PROGRAM PresenceSimulation
VAR
	
	fbWeeklyTimeSwitch	:FB_WeeklyTimeSwitch;
	fbSceneLight		:FB_IoT_Switch(P_IoT_Com.fbIoT_ComClient,0);
	CTU					:CTU;
	TON					:ARRAY[1..55] OF TON;
	TP					:ARRAY[1..55] OF TP;
	
	bAnwesenheit_Tag_1_aktivieren: BOOL;
	bAnwesenheit_Tag_2_aktivieren: BOOL;
	bAnwesenheit_Tag_3_aktivieren: BOOL;
	bAnwesenheit_Tag_4_aktivieren: BOOL;
	bAnwesenheit_Tag_5_aktivieren: BOOL;
	
	bAnwesenheit_1_Beleuchtung_1: BOOL;
	bAnwesenheit_1_Beleuchtung_2: BOOL;
	bAnwesenheit_1_Beleuchtung_3: BOOL;
	bAnwesenheit_1_Beleuchtung_4: BOOL;
	bAnwesenheit_1_Beleuchtung_5: BOOL;
	
	bAnwesenheit_2_Beleuchtung_1: BOOL;
	bAnwesenheit_2_Beleuchtung_2: BOOL;
	bAnwesenheit_2_Beleuchtung_3: BOOL;
	bAnwesenheit_2_Beleuchtung_4: BOOL;
	bAnwesenheit_2_Beleuchtung_5: BOOL;
	
	bAnwesenheit_3_Beleuchtung_1: BOOL;
	bAnwesenheit_3_Beleuchtung_2: BOOL;
	bAnwesenheit_3_Beleuchtung_3: BOOL;
	bAnwesenheit_3_Beleuchtung_4: BOOL;
	bAnwesenheit_3_Beleuchtung_5: BOOL;
	
	bAnwesenheit_4_Beleuchtung_1: BOOL;
	bAnwesenheit_4_Beleuchtung_2: BOOL;
	bAnwesenheit_4_Beleuchtung_3: BOOL;
	bAnwesenheit_4_Beleuchtung_4: BOOL;
	bAnwesenheit_4_Beleuchtung_5: BOOL;
	
	bAnwesenheit_5_Beleuchtung_1: BOOL;
	bAnwesenheit_5_Beleuchtung_2: BOOL;
	bAnwesenheit_5_Beleuchtung_3: BOOL;
	bAnwesenheit_5_Beleuchtung_4: BOOL;
	bAnwesenheit_5_Beleuchtung_5: BOOL;
END_VAR
VAR // added by the converter: edge detectors and wires of the graphical bodies
    _w1 : BOOL;
END_VAR

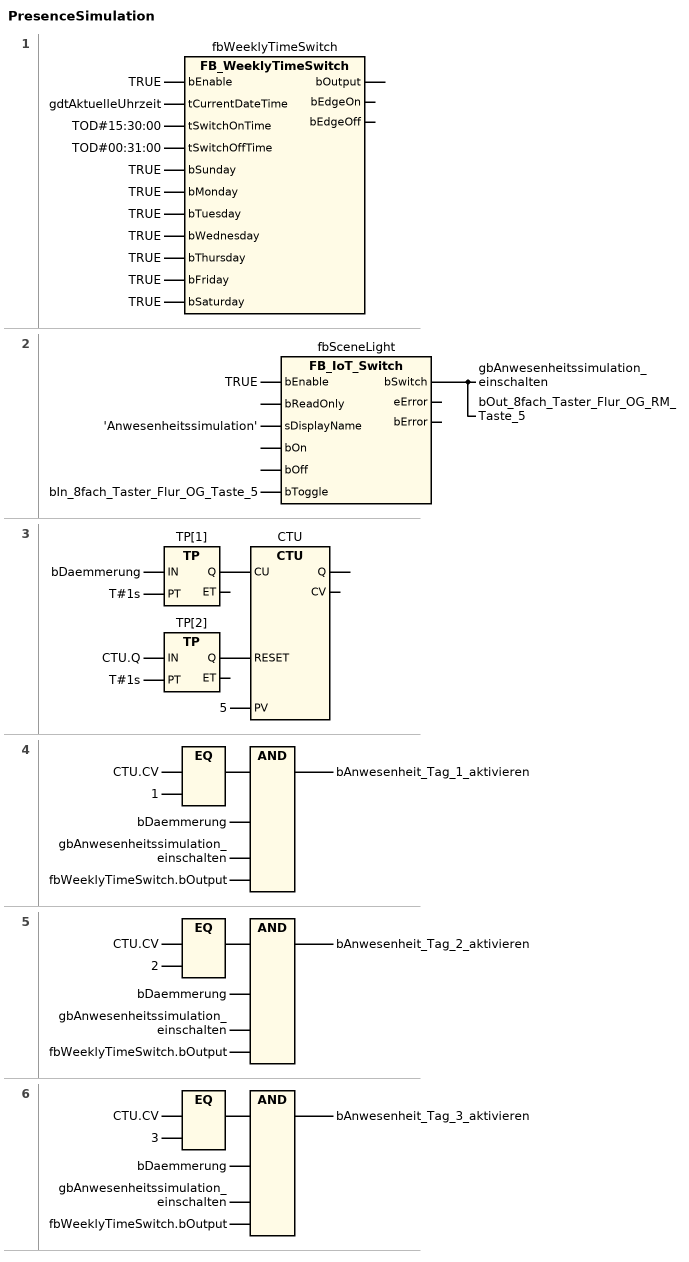
// NETWORK 1
fbWeeklyTimeSwitch(
    bEnable := TRUE,
    tCurrentDateTime := gdtAktuelleUhrzeit,
    tSwitchOnTime := TOD#15:30:00,
    tSwitchOffTime := TOD#00:31:00,
    bSunday := TRUE,
    bMonday := TRUE,
    bTuesday := TRUE,
    bWednesday := TRUE,
    bThursday := TRUE,
    bFriday := TRUE,
    bSaturday := TRUE); // FB_WeeklyTimeSwitch

// NETWORK 2
fbSceneLight(
    bEnable := TRUE,
    sDisplayName := 'Anwesenheitssimulation',
    bToggle := bIn_8fach_Taster_Flur_OG_Taste_5); // FB_IoT_Switch
gbAnwesenheitssimulation_einschalten := fbSceneLight.bSwitch;
bOut_8fach_Taster_Flur_OG_RM_Taste_5 := fbSceneLight.bSwitch;

// NETWORK 3
TP[1](IN := bDaemmerung, PT := T#1s); // TP
_w1 := TP[1].Q;
TP[2](IN := CTU.Q, PT := T#1s); // TP
CTU(CU := _w1, RESET := TP[2].Q, PV := 5);

// NETWORK 4
bAnwesenheit_Tag_1_aktivieren := CTU.CV = 1 AND bDaemmerung AND gbAnwesenheitssimulation_einschalten AND fbWeeklyTimeSwitch.bOutput;

// NETWORK 5
bAnwesenheit_Tag_2_aktivieren := CTU.CV = 2 AND bDaemmerung AND gbAnwesenheitssimulation_einschalten AND fbWeeklyTimeSwitch.bOutput;

// NETWORK 6
bAnwesenheit_Tag_3_aktivieren := CTU.CV = 3 AND bDaemmerung AND gbAnwesenheitssimulation_einschalten AND fbWeeklyTimeSwitch.bOutput;

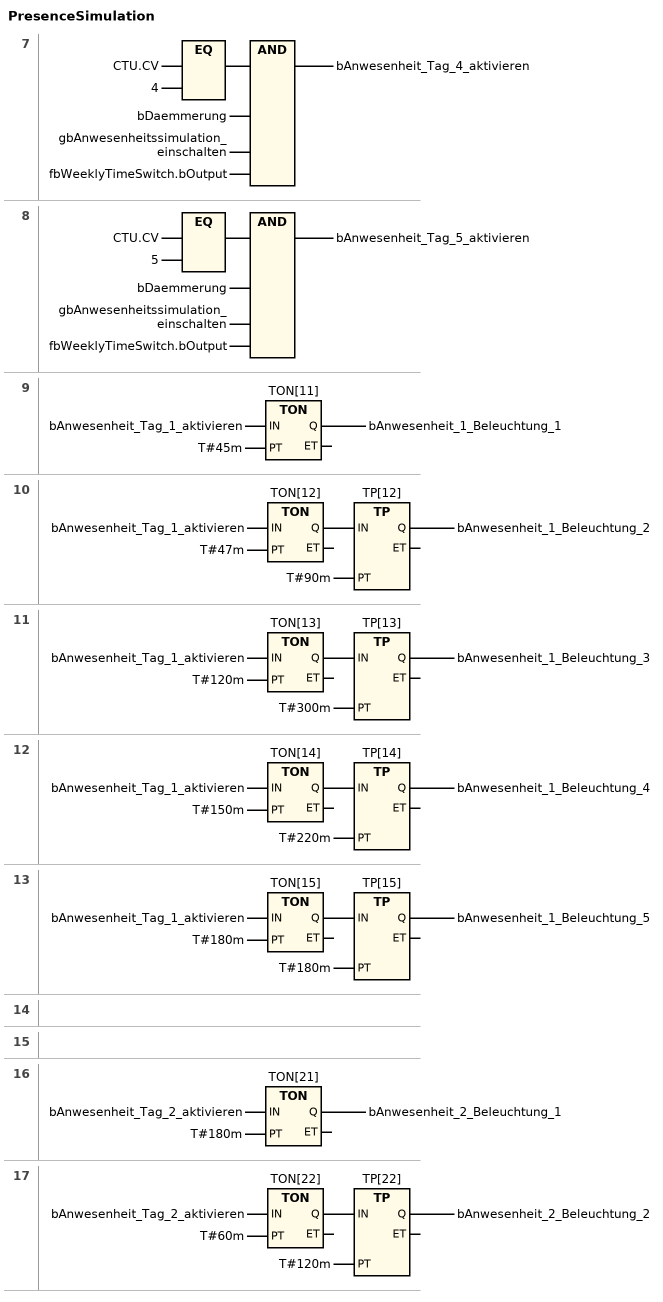
// NETWORK 7
bAnwesenheit_Tag_4_aktivieren := CTU.CV = 4 AND bDaemmerung AND gbAnwesenheitssimulation_einschalten AND fbWeeklyTimeSwitch.bOutput;

// NETWORK 8
bAnwesenheit_Tag_5_aktivieren := CTU.CV = 5 AND bDaemmerung AND gbAnwesenheitssimulation_einschalten AND fbWeeklyTimeSwitch.bOutput;

// NETWORK 9
TON[11](IN := bAnwesenheit_Tag_1_aktivieren, PT := T#45m); // TON
bAnwesenheit_1_Beleuchtung_1 := TON[11].Q;

// NETWORK 10
TON[12](IN := bAnwesenheit_Tag_1_aktivieren, PT := T#47m); // TON
TP[12](IN := TON[12].Q, PT := T#90m); // TP
bAnwesenheit_1_Beleuchtung_2 := TP[12].Q;

// NETWORK 11
TON[13](IN := bAnwesenheit_Tag_1_aktivieren, PT := T#120m); // TON
TP[13](IN := TON[13].Q, PT := T#300m); // TP
bAnwesenheit_1_Beleuchtung_3 := TP[13].Q;

// NETWORK 12
TON[14](IN := bAnwesenheit_Tag_1_aktivieren, PT := T#150m); // TON
TP[14](IN := TON[14].Q, PT := T#220m); // TP
bAnwesenheit_1_Beleuchtung_4 := TP[14].Q;

// NETWORK 13
TON[15](IN := bAnwesenheit_Tag_1_aktivieren, PT := T#180m); // TON
TP[15](IN := TON[15].Q, PT := T#180m); // TP
bAnwesenheit_1_Beleuchtung_5 := TP[15].Q;

// NETWORK 14

// NETWORK 15

// NETWORK 16
TON[21](IN := bAnwesenheit_Tag_2_aktivieren, PT := T#180m); // TON
bAnwesenheit_2_Beleuchtung_1 := TON[21].Q;

// NETWORK 17
TON[22](IN := bAnwesenheit_Tag_2_aktivieren, PT := T#60m); // TON
TP[22](IN := TON[22].Q, PT := T#120m); // TP
bAnwesenheit_2_Beleuchtung_2 := TP[22].Q;

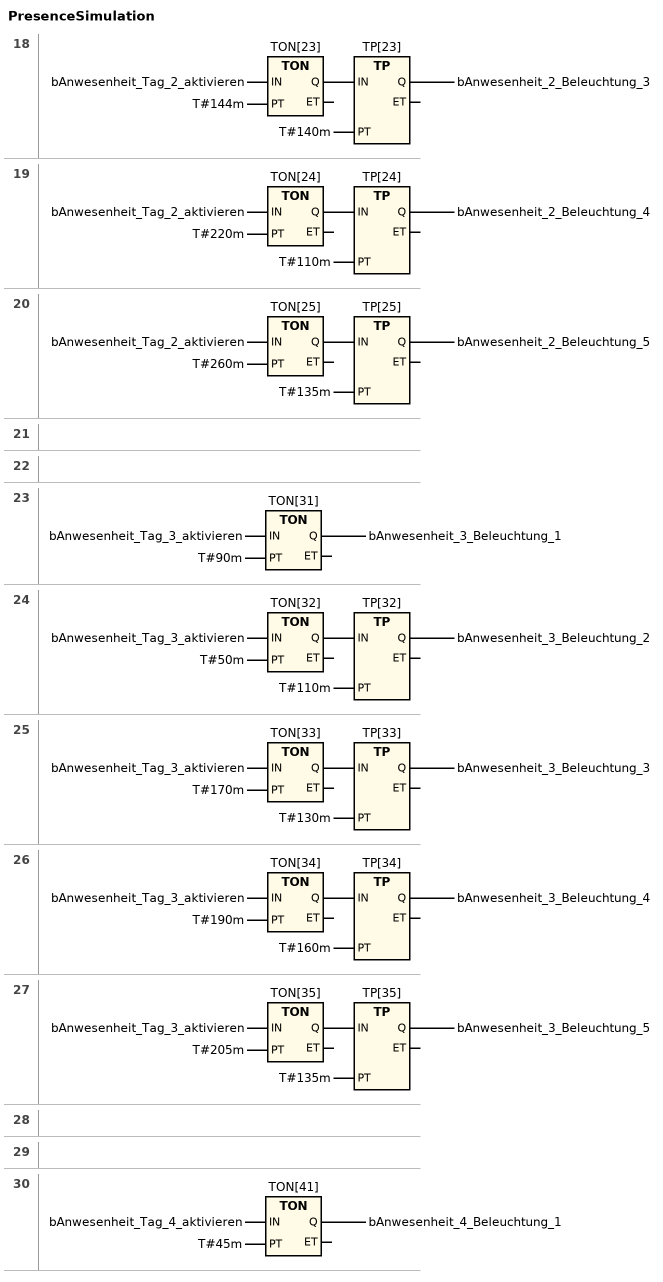
// NETWORK 18
TON[23](IN := bAnwesenheit_Tag_2_aktivieren, PT := T#144m); // TON
TP[23](IN := TON[23].Q, PT := T#140m); // TP
bAnwesenheit_2_Beleuchtung_3 := TP[23].Q;

// NETWORK 19
TON[24](IN := bAnwesenheit_Tag_2_aktivieren, PT := T#220m); // TON
TP[24](IN := TON[24].Q, PT := T#110m); // TP
bAnwesenheit_2_Beleuchtung_4 := TP[24].Q;

// NETWORK 20
TON[25](IN := bAnwesenheit_Tag_2_aktivieren, PT := T#260m); // TON
TP[25](IN := TON[25].Q, PT := T#135m); // TP
bAnwesenheit_2_Beleuchtung_5 := TP[25].Q;

// NETWORK 21

// NETWORK 22

// NETWORK 23
TON[31](IN := bAnwesenheit_Tag_3_aktivieren, PT := T#90m); // TON
bAnwesenheit_3_Beleuchtung_1 := TON[31].Q;

// NETWORK 24
TON[32](IN := bAnwesenheit_Tag_3_aktivieren, PT := T#50m); // TON
TP[32](IN := TON[32].Q, PT := T#110m); // TP
bAnwesenheit_3_Beleuchtung_2 := TP[32].Q;

// NETWORK 25
TON[33](IN := bAnwesenheit_Tag_3_aktivieren, PT := T#170m); // TON
TP[33](IN := TON[33].Q, PT := T#130m); // TP
bAnwesenheit_3_Beleuchtung_3 := TP[33].Q;

// NETWORK 26
TON[34](IN := bAnwesenheit_Tag_3_aktivieren, PT := T#190m); // TON
TP[34](IN := TON[34].Q, PT := T#160m); // TP
bAnwesenheit_3_Beleuchtung_4 := TP[34].Q;

// NETWORK 27
TON[35](IN := bAnwesenheit_Tag_3_aktivieren, PT := T#205m); // TON
TP[35](IN := TON[35].Q, PT := T#135m); // TP
bAnwesenheit_3_Beleuchtung_5 := TP[35].Q;

// NETWORK 28

// NETWORK 29

// NETWORK 30
TON[41](IN := bAnwesenheit_Tag_4_aktivieren, PT := T#45m); // TON
bAnwesenheit_4_Beleuchtung_1 := TON[41].Q;

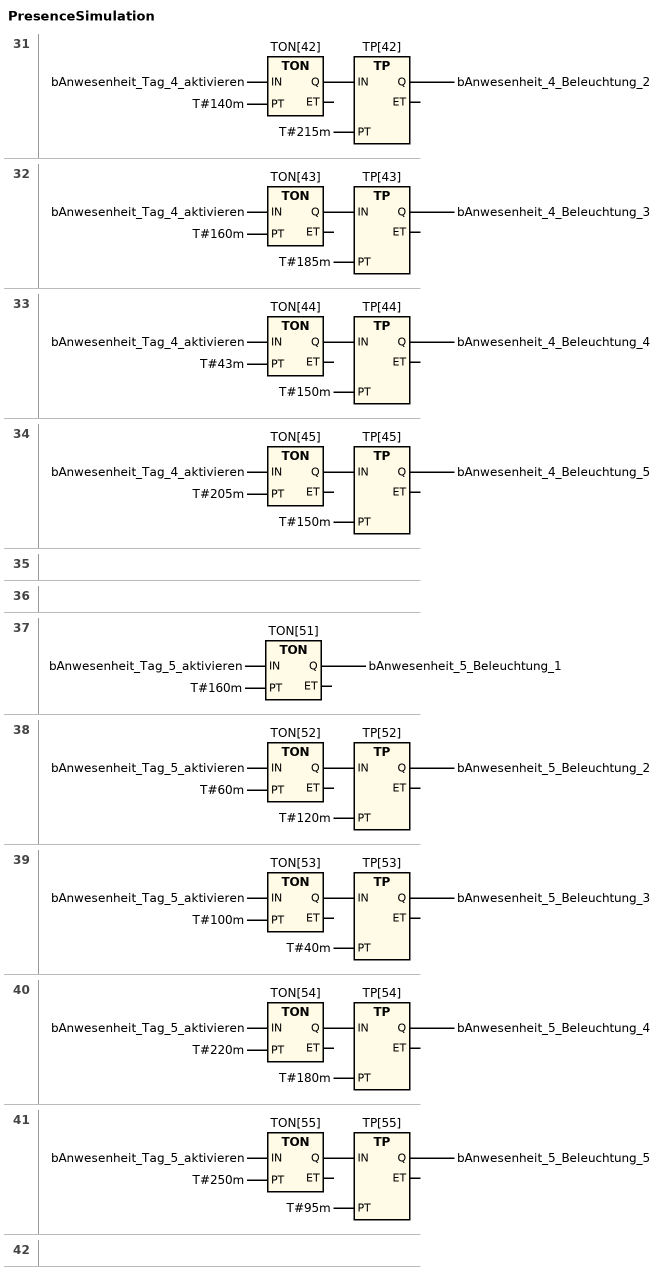
// NETWORK 31
TON[42](IN := bAnwesenheit_Tag_4_aktivieren, PT := T#140m); // TON
TP[42](IN := TON[42].Q, PT := T#215m); // TP
bAnwesenheit_4_Beleuchtung_2 := TP[42].Q;

// NETWORK 32
TON[43](IN := bAnwesenheit_Tag_4_aktivieren, PT := T#160m); // TON
TP[43](IN := TON[43].Q, PT := T#185m); // TP
bAnwesenheit_4_Beleuchtung_3 := TP[43].Q;

// NETWORK 33
TON[44](IN := bAnwesenheit_Tag_4_aktivieren, PT := T#43m); // TON
TP[44](IN := TON[44].Q, PT := T#150m); // TP
bAnwesenheit_4_Beleuchtung_4 := TP[44].Q;

// NETWORK 34
TON[45](IN := bAnwesenheit_Tag_4_aktivieren, PT := T#205m); // TON
TP[45](IN := TON[45].Q, PT := T#150m); // TP
bAnwesenheit_4_Beleuchtung_5 := TP[45].Q;

// NETWORK 35

// NETWORK 36

// NETWORK 37
TON[51](IN := bAnwesenheit_Tag_5_aktivieren, PT := T#160m); // TON
bAnwesenheit_5_Beleuchtung_1 := TON[51].Q;

// NETWORK 38
TON[52](IN := bAnwesenheit_Tag_5_aktivieren, PT := T#60m); // TON
TP[52](IN := TON[52].Q, PT := T#120m); // TP
bAnwesenheit_5_Beleuchtung_2 := TP[52].Q;

// NETWORK 39
TON[53](IN := bAnwesenheit_Tag_5_aktivieren, PT := T#100m); // TON
TP[53](IN := TON[53].Q, PT := T#40m); // TP
bAnwesenheit_5_Beleuchtung_3 := TP[53].Q;

// NETWORK 40
TON[54](IN := bAnwesenheit_Tag_5_aktivieren, PT := T#220m); // TON
TP[54](IN := TON[54].Q, PT := T#180m); // TP
bAnwesenheit_5_Beleuchtung_4 := TP[54].Q;

// NETWORK 41
TON[55](IN := bAnwesenheit_Tag_5_aktivieren, PT := T#250m); // TON
TP[55](IN := TON[55].Q, PT := T#95m); // TP
bAnwesenheit_5_Beleuchtung_5 := TP[55].Q;

// NETWORK 42

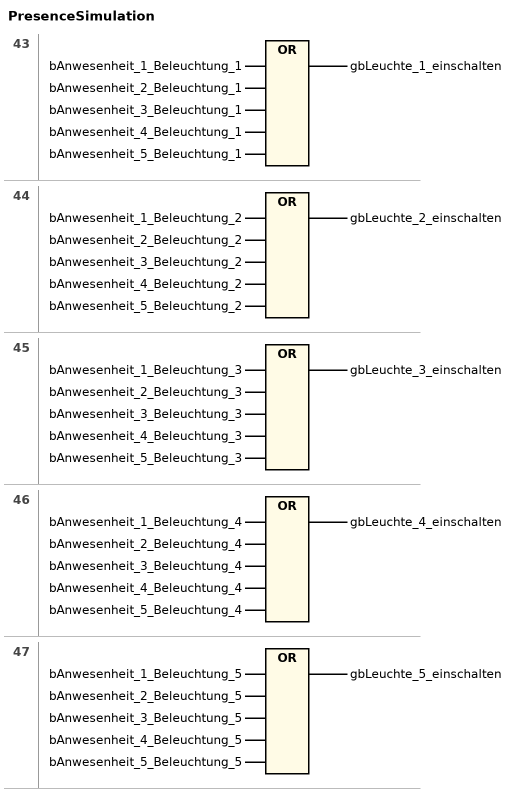
// NETWORK 43
gbLeuchte_1_einschalten := bAnwesenheit_1_Beleuchtung_1 OR bAnwesenheit_2_Beleuchtung_1 OR bAnwesenheit_3_Beleuchtung_1 OR bAnwesenheit_4_Beleuchtung_1 OR bAnwesenheit_5_Beleuchtung_1;

// NETWORK 44
gbLeuchte_2_einschalten := bAnwesenheit_1_Beleuchtung_2 OR bAnwesenheit_2_Beleuchtung_2 OR bAnwesenheit_3_Beleuchtung_2 OR bAnwesenheit_4_Beleuchtung_2 OR bAnwesenheit_5_Beleuchtung_2;

// NETWORK 45
gbLeuchte_3_einschalten := bAnwesenheit_1_Beleuchtung_3 OR bAnwesenheit_2_Beleuchtung_3 OR bAnwesenheit_3_Beleuchtung_3 OR bAnwesenheit_4_Beleuchtung_3 OR bAnwesenheit_5_Beleuchtung_3;

// NETWORK 46
gbLeuchte_4_einschalten := bAnwesenheit_1_Beleuchtung_4 OR bAnwesenheit_2_Beleuchtung_4 OR bAnwesenheit_3_Beleuchtung_4 OR bAnwesenheit_4_Beleuchtung_4 OR bAnwesenheit_5_Beleuchtung_4;

// NETWORK 47
gbLeuchte_5_einschalten := bAnwesenheit_1_Beleuchtung_5 OR bAnwesenheit_2_Beleuchtung_5 OR bAnwesenheit_3_Beleuchtung_5 OR bAnwesenheit_4_Beleuchtung_5 OR bAnwesenheit_5_Beleuchtung_5;

END_PROGRAM

(* stored: Version 1.1.0.1, ProductVersion 3.1.4024.11
   POU PresenceSimulation: Id {533ade04-e697-40da-8af7-820fe56d5ca8}, SpecialFunc None *)
